(* IEC 61131-3 sources: axftcmlib/src/Axis/SpeedAxis, 4 files *)

(* ---- itfSpeedAxis.st ---- *)
USING Simatic.Ax.Commands;

NAMESPACE Simatic.Ax.axftcmlib.Motion

    INTERFACE itfSpeedAxis EXTENDS itfAxis

    METHOD MoveVelocity : itfCommand
        VAR_INPUT
            Velocity : LReal := 100.0;
            Direction : Direction := Direction#PositiveDirection;
        END_VAR
    END_METHOD

    METHOD Stop : itfCommand
    END_METHOD

END_INTERFACE

END_NAMESPACE

(* ---- commandMoveVelovity.st ---- *)
USING Simatic.Ax.Commands;

NAMESPACE Simatic.Ax.axftcmlib.Motion

    CLASS INTERNAL commandMoveVelovity
        EXTENDS ExecuteCommand
        VAR
            _AxisRef : REF_TO TO_SpeedAxis;
            _velocity : LReal;
            _direction : Direction;
        END_VAR

        METHOD PUBLIC Start : itfCommand
            VAR_INPUT
                AxisRef : REF_TO TO_SpeedAxis;
                Velocity : LReal  := LReal#100.0;
                Direction : Direction := Direction#PositiveDirection;
            END_VAR
            _AxisRef := AxisRef;
            _velocity := Velocity;
            _direction := Direction;
            THIS.ExecuteWithRisingEdge();
            Start := THIS;
        END_METHOD

        METHOD PROTECTED OVERRIDE Execute
            IF (NOT _AxisRef^.isPowerdOn) THEN
                THIS.SetError(WORD#16#8001);
            ELSE
                ;
            END_IF;
        END_METHOD

        METHOD PROTECTED OVERRIDE SetExecute
            VAR_INPUT
                exec : BOOL;
            END_VAR
            IF (NOT _AxisRef^.isPowerdOn) THEN
                THIS.SetError(WORD#16#8001);
            ELSE
                _AxisRef^.Run(TRUE);
                _AxisRef^.Velocity := _velocity;
                _AxisRef^.Direction := _direction;
            END_IF;

        END_METHOD
    END_CLASS

END_NAMESPACE

(* ---- commandStop.st ---- *)
USING Simatic.Ax.Commands;

NAMESPACE Simatic.Ax.axftcmlib.Motion

    CLASS INTERNAL commandStop
        EXTENDS ExecuteCommand
        VAR
            _AxisRef : REF_TO TO_SpeedAxis;
        END_VAR

        METHOD PUBLIC Start : itfCommand
            VAR_INPUT
                AxisRef : REF_TO TO_SpeedAxis;
            END_VAR
            _AxisRef := AxisRef;
            THIS.ExecuteWithRisingEdge();
            Start := THIS;
        END_METHOD

        METHOD PROTECTED OVERRIDE Execute
            ;
        END_METHOD

        METHOD PROTECTED OVERRIDE SetExecute
            VAR_INPUT
                exec : BOOL;
            END_VAR

            _AxisRef^.Run(FALSE);
            THIS.SetDone();

        END_METHOD
    END_CLASS

END_NAMESPACE

(* ---- SpeedAxis.st ---- *)
USING Simatic.Ax.Commands;

NAMESPACE Simatic.Ax.axftcmlib.Motion

    CLASS SpeedAxis
        EXTENDS SpeedAxisImpl

        METHOD PUBLIC Attach : BOOL
            VAR_INPUT
                axis : REF_TO TO_SpeedAxis;
            END_VAR
            _SpeedAxisRef := axis;
            SUPER.Attach(axis);
            Attach := THIS.IsAttached();
        END_METHOD
    END_CLASS

    CLASS INTERNAL SpeedAxisImpl
        EXTENDS AxisBase
        IMPLEMENTS itfSpeedAxis
        VAR PROTECTED
            _SpeedAxisRef : REF_TO TO_SpeedAxis;
            _commandMoveVelocity : commandMoveVelovity;
            _commandStop : commandStop;
        END_VAR

        METHOD PUBLIC MoveVelocity : itfCommand
            VAR_INPUT
                Velocity : LREAL := 100.0;
                Direction : Direction := Direction#PositiveDirection;
            END_VAR
            MoveVelocity := _commandMoveVelocity.Start(AxisRef := _SpeedAxisRef, Velocity := Velocity, Direction := Direction);
        END_METHOD

        METHOD PUBLIC Stop : itfCommand
            Stop := _commandStop.Start(AxisRef := _SpeedAxisRef);
        END_METHOD

        METHOD PROTECTED OVERRIDE MakeAxisAbstract
            ;
        END_METHOD
    END_CLASS

END_NAMESPACE
